(* IEC 61131-3 sources: ST2CPP/examples/projects/robot_arm, 8 files *)

(* ---- math_utils.st ---- *)
(* math_utils.st — 数学工具函数 *)

FUNCTION DEG_TO_RAD : REAL
    VAR_INPUT DEG : REAL; END_VAR
    DEG_TO_RAD := DEG * 3.14159265 / 180.0;
END_FUNCTION

FUNCTION RAD_TO_DEG : REAL
    VAR_INPUT RAD : REAL; END_VAR
    RAD_TO_DEG := RAD * 180.0 / 3.14159265;
END_FUNCTION

FUNCTION CLAMP_REAL : REAL
    VAR_INPUT VAL : REAL; MN : REAL; MX : REAL; END_VAR
    IF VAL > MX THEN
        CLAMP_REAL := MX;
    ELSIF VAL < MN THEN
        CLAMP_REAL := MN;
    ELSE
        CLAMP_REAL := VAL;
    END_IF;
END_FUNCTION

FUNCTION CLAMP_DINT : DINT
    VAR_INPUT VAL : DINT; MN : DINT; MX : DINT; END_VAR
    IF VAL > MX THEN
        CLAMP_DINT := MX;
    ELSIF VAL < MN THEN
        CLAMP_DINT := MN;
    ELSE
        CLAMP_DINT := VAL;
    END_IF;
END_FUNCTION

FUNCTION ABS_REAL : REAL
    VAR_INPUT X : REAL; END_VAR
    IF X < 0.0 THEN
        ABS_REAL := 0.0 - X;
    ELSE
        ABS_REAL := X;
    END_IF;
END_FUNCTION

FUNCTION ABS_DINT : DINT
    VAR_INPUT X : DINT; END_VAR
    IF X < 0 THEN
        ABS_DINT := 0 - X;
    ELSE
        ABS_DINT := X;
    END_IF;
END_FUNCTION

FUNCTION SIGN_REAL : REAL
    VAR_INPUT X : REAL; END_VAR
    IF X > 0.0 THEN
        SIGN_REAL := 1.0;
    ELSIF X < 0.0 THEN
        SIGN_REAL := -1.0;
    ELSE
        SIGN_REAL := 0.0;
    END_IF;
END_FUNCTION

(* 简单梯形速度规划：返回当前周期的目标位置 *)
FUNCTION TRAPZ_POSITION : DINT
    VAR_INPUT
        POS_START   : DINT;     (* 起始位置 *)
        POS_END     : DINT;     (* 目标位置 *)
        VEL_MAX     : DINT;     (* 最大速度 *)
        ACC_MAX     : DINT;     (* 最大加速度 *)
        TIME_MS     : DINT;     (* 已用时间 ms *)
        TOTAL_MS    : DINT;     (* 总时间 ms *)
    END_VAR
    VAR
        DIST        : DINT;
        SIGN_DIR    : DINT;
        ACCEL_TIME  : DINT;
        cruise_time : DINT;
        pos         : DINT;
    END_VAR

    DIST := ABS_DINT(POS_END - POS_START);
    IF POS_END >= POS_START THEN
        SIGN_DIR := 1;
    ELSE
        SIGN_DIR := -1;
    END_IF;

    IF VEL_MAX <= 0 OR ACC_MAX <= 0 OR TOTAL_MS <= 0 THEN
        TRAPZ_POSITION := POS_START;
        RETURN;
    END_IF;

    ACCEL_TIME := VEL_MAX * 1000 / ACC_MAX;
    IF ACCEL_TIME > TOTAL_MS / 2 THEN
        ACCEL_TIME := TOTAL_MS / 2;
    END_IF;

    cruise_time := TOTAL_MS - 2 * ACCEL_TIME;

    IF TIME_MS < ACCEL_TIME THEN
        (* 加速段 *)
        pos := POS_START + SIGN_DIR * ACC_MAX * TIME_MS * TIME_MS / 2000000;
    ELSIF TIME_MS < ACCEL_TIME + cruise_time THEN
        (* 匀速段 *)
        pos := POS_START + SIGN_DIR * (VEL_MAX * ACCEL_TIME / 1000 + VEL_MAX * (TIME_MS - ACCEL_TIME) / 1000);
    ELSIF TIME_MS < TOTAL_MS THEN
        (* 减速段 *)
        pos := POS_END - SIGN_DIR * ACC_MAX * (TOTAL_MS - TIME_MS) * (TOTAL_MS - TIME_MS) / 2000000;
    ELSE
        pos := POS_END;
    END_IF;

    TRAPZ_POSITION := pos;
END_FUNCTION

(* 两点间距离 *)
FUNCTION DISTANCE_3D : REAL
    VAR_INPUT A : POSE_3D; B : POSE_3D; END_VAR
    VAR DX : REAL; DY : REAL; DZ : REAL; END_VAR
    DX := B.X - A.X;
    DY := B.Y - A.Y;
    DZ := B.Z - A.Z;
    DISTANCE_3D := (DX * DX + DY * DY + DZ * DZ);
END_FUNCTION

(* ---- motion_planner.st ---- *)
(* motion_planner.st — 关节空间运动规划器 *)

FUNCTION_BLOCK JOINT_PLANNER
    VAR_INPUT
        TARGET_J    : JOINT_WAYPOINT;   (* 目标关节角度 *)
        SPEED_PCT   : REAL;             (* 速度百分比 0-100 *)
        START       : BOOL;             (* 启动运动 *)
        STOP        : BOOL;             (* 停止运动 *)
        ABORT       : BOOL;             (* 紧急终止 *)
    END_VAR
    VAR_OUTPUT
        CMD_J       : JOINT_WAYPOINT;   (* 当前周期命令 *)
        DONE        : BOOL;             (* 运动完成 *)
        MOVING      : BOOL;             (* 运动中 *)
        PROGRESS    : REAL;             (* 进度 0-100 *)
        ERROR       : BOOL;
        ERROR_CODE  : INT;
    END_VAR
    VAR
        STATE       : INT := 0;         (* 0=Idle, 1=Planning, 2=Moving, 3=Done *)
        START_J     : JOINT_WAYPOINT;   (* 起始关节角度 *)
        TIME_MS     : DINT := 0;
        TOTAL_MS    : DINT := 0;
        SPEED_SCALE : REAL;
        I           : INT;
        DUR         : DINT;
        MAX_DUR     : DINT;
    END_VAR

    IF ABORT THEN
        STATE := 0;
        MOVING := FALSE;
        DONE := FALSE;
        ERROR := TRUE;
        ERROR_CODE := 99;
        RETURN;
    END_IF;

    IF STOP AND STATE = 2 THEN
        STATE := 0;
        MOVING := FALSE;
        DONE := FALSE;
        RETURN;
    END_IF;

    CASE STATE OF
        0:
            (* Idle *)
            DONE := FALSE;
            MOVING := FALSE;
            PROGRESS := 0.0;
            ERROR := FALSE;
            ERROR_CODE := 0;
            IF START THEN
                STATE := 1;
                TIME_MS := 0;
                MAX_DUR := 0;
                SPEED_SCALE := SPEED_PCT / 100.0;
                IF SPEED_SCALE < 0.1 THEN
                    SPEED_SCALE := 0.1;
                END_IF;
                IF SPEED_SCALE > 1.0 THEN
                    SPEED_SCALE := 1.0;
                END_IF;
            END_IF;

        1:
            (* Planning — 计算运动时间 *)
            (* J1 *)
            DUR := ABS_DINT(TARGET_J.J1 * 100);
            IF DUR > MAX_DUR THEN MAX_DUR := DUR; END_IF;
            (* J2 *)
            DUR := ABS_DINT(TARGET_J.J2 * 100);
            IF DUR > MAX_DUR THEN MAX_DUR := DUR; END_IF;
            (* J3 *)
            DUR := ABS_DINT(TARGET_J.J3 * 100);
            IF DUR > MAX_DUR THEN MAX_DUR := DUR; END_IF;
            (* J4 *)
            DUR := ABS_DINT(TARGET_J.J4 * 100);
            IF DUR > MAX_DUR THEN MAX_DUR := DUR; END_IF;
            (* J5 *)
            DUR := ABS_DINT(TARGET_J.J5 * 100);
            IF DUR > MAX_DUR THEN MAX_DUR := DUR; END_IF;
            (* J6 *)
            DUR := ABS_DINT(TARGET_J.J6 * 100);
            IF DUR > MAX_DUR THEN MAX_DUR := DUR; END_IF;

            TOTAL_MS := MAX_DUR * 10 / SPEED_SCALE + 500;
            IF TOTAL_MS < 100 THEN TOTAL_MS := 100; END_IF;
            IF TOTAL_MS > 5000 THEN TOTAL_MS := 5000; END_IF;

            START_J.J1 := CMD_J.J1;
            START_J.J2 := CMD_J.J2;
            START_J.J3 := CMD_J.J3;
            START_J.J4 := CMD_J.J4;
            START_J.J5 := CMD_J.J5;
            START_J.J6 := CMD_J.J6;

            STATE := 2;
            MOVING := TRUE;

        2:
            (* Moving — 每个周期更新 *)
            TIME_MS := TIME_MS + 10;

            CMD_J.J1 := TRAPZ_POSITION(START_J.J1, TARGET_J.J1, 1000, 200, TIME_MS, TOTAL_MS);
            CMD_J.J2 := TRAPZ_POSITION(START_J.J2, TARGET_J.J2, 800, 150, TIME_MS, TOTAL_MS);
            CMD_J.J3 := TRAPZ_POSITION(START_J.J3, TARGET_J.J3, 800, 150, TIME_MS, TOTAL_MS);
            CMD_J.J4 := TRAPZ_POSITION(START_J.J4, TARGET_J.J4, 1200, 300, TIME_MS, TOTAL_MS);
            CMD_J.J5 := TRAPZ_POSITION(START_J.J5, TARGET_J.J5, 1200, 300, TIME_MS, TOTAL_MS);
            CMD_J.J6 := TRAPZ_POSITION(START_J.J6, TARGET_J.J6, 1500, 400, TIME_MS, TOTAL_MS);

            IF TOTAL_MS > 0 THEN
                PROGRESS := TIME_MS * 100.0 / TOTAL_MS;
            END_IF;
            IF PROGRESS > 100.0 THEN PROGRESS := 100.0; END_IF;

            IF TIME_MS >= TOTAL_MS THEN
                CMD_J.J1 := TARGET_J.J1;
                CMD_J.J2 := TARGET_J.J2;
                CMD_J.J3 := TARGET_J.J3;
                CMD_J.J4 := TARGET_J.J4;
                CMD_J.J5 := TARGET_J.J5;
                CMD_J.J6 := TARGET_J.J6;
                STATE := 3;
                MOVING := FALSE;
                DONE := TRUE;
                PROGRESS := 100.0;
            END_IF;

        3:
            (* Done *)
            MOVING := FALSE;
            IF NOT START THEN
                STATE := 0;
                DONE := FALSE;
            END_IF;
    END_CASE;
END_FUNCTION_BLOCK

(* ---- robot_ctrl.st ---- *)
(* robot_ctrl.st — 6轴机械臂主控制器 *)

FUNCTION_BLOCK ROBOT_CTRL
    VAR_INPUT
        START           : BOOL;
        STOP            : BOOL;
        HOME_CMD        : BOOL;
        AUTO_MODE       : BOOL;
        TEACH_MODE      : BOOL;
        SPEED_OVERRIDE  : REAL;          (* 速度倍率 0-100% *)
    END_VAR
    VAR_OUTPUT
        STATE_OUT       : INT;           (* 0=Disabled, 1=Idle, 2=Running, 3=Homing, 4=Error *)
        FAULT           : BOOL;
        FAULT_CODE      : INT;
        HOME_DONE       : BOOL;
        STEP_NUM        : INT;
        CYCLE_COUNT     : DINT;
    END_VAR
    VAR
        (* 6轴伺服 *)
        Srv             : ARRAY[0..5] OF SERVO_CTRL;

        (* 运动规划器 *)
        Planner         : JOINT_PLANNER;

        (* 安全监控 *)
        SafetyMon       : SAFETY_MONITOR;

        (* 关节限位 [轴号][0=下限,1=上限] *)
        JOINT_LIM       : ARRAY[0..5, 0..1] OF DINT;

        (* 伺服状态 *)
        SrvReady        : ARRAY[0..5] OF BOOL;
        SrvFaultArr     : ARRAY[0..5] OF BOOL;
        ActPosArr       : ARRAY[0..5] OF DINT;

        (* 工序步 *)
        PROG_STEP       : INT := 0;
        STEP_ACTIVE     : BOOL := FALSE;
        ALL_DONE        : BOOL := FALSE;

        (* 工序定义：抓取-放置 *)
        GRAB_POS        : JOINT_WAYPOINT := (J1 := 0.0, J2 := -45.0, J3 := 90.0, J4 := 0.0, J5 := 45.0, J6 := 0.0, SPEED := 50.0, DWELL_MS := 500);
        PRE_GRAB_POS    : JOINT_WAYPOINT := (J1 := 0.0, J2 := -20.0, J3 := 45.0, J4 := 0.0, J5 := 20.0, J6 := 0.0, SPEED := 30.0, DWELL_MS := 200);
        HOME_POS        : JOINT_WAYPOINT := (J1 := 0.0, J2 := 0.0, J3 := 0.0, J4 := 0.0, J5 := 0.0, J6 := 0.0, SPEED := 20.0, DWELL_MS := 0);
        PLACE_POS       : JOINT_WAYPOINT := (J1 := 90.0, J2 := -30.0, J3 := 60.0, J4 := 0.0, J5 := 30.0, J6 := 90.0, SPEED := 40.0, DWELL_MS := 300);
        RETRACT_POS     : JOINT_WAYPOINT := (J1 := 90.0, J2 := 0.0, J3 := 0.0, J4 := 0.0, J5 := 0.0, J6 := 0.0, SPEED := 50.0, DWELL_MS := 200);

        (* 辅助 *)
        I               : INT;
        SRV_EN          : ARRAY[0..5] OF BOOL;
        START_PREV      : BOOL := FALSE;
        TRIG_START      : BOOL;
        HOME_PREV       : BOOL := FALSE;
        TRIG_HOME       : BOOL;
        DWELL_TIMER     : INT := 0;
        DWELL_TARGET    : INT := 0;
    END_VAR

    TRIG_START := START AND NOT START_PREV;
    START_PREV := START;
    TRIG_HOME := HOME_CMD AND NOT HOME_PREV;
    HOME_PREV := HOME_CMD;

    (* ─── 关节限位初始化 ─── *)
    JOINT_LIM[0, 0] := -170000;
    JOINT_LIM[0, 1] := 170000;
    JOINT_LIM[1, 0] := -120000;
    JOINT_LIM[1, 1] := 120000;
    JOINT_LIM[2, 0] := -150000;
    JOINT_LIM[2, 1] := 150000;
    JOINT_LIM[3, 0] := -180000;
    JOINT_LIM[3, 1] := 180000;
    JOINT_LIM[4, 0] := -120000;
    JOINT_LIM[4, 1] := 120000;
    JOINT_LIM[5, 0] := -360000;
    JOINT_LIM[5, 1] := 360000;

    (* ─── 速度倍率钳位 ─── *)
    SPEED_OVERRIDE := CLAMP_REAL(SPEED_OVERRIDE, 5.0, 100.0);

    (* ─── 使能所有伺服 ─── *)
    FOR I := 0 TO 5 DO
        SRV_EN[I] := START AND NOT FAULT;
    END_FOR;

    (* ─── 执行伺服控制 ─── *)
    FOR I := 0 TO 5 DO
        Srv[I](
            AXIS_ID := I,
            CMD_POSITION := Planner.CMD_J.J1,
            CMD_MODE := 0,
            ENABLE := SRV_EN[I],
            HOME_CMD := TRIG_HOME,
            RESET_CMD := FALSE,
            VEL_LIMIT := 2000,
            TORQ_LIMIT := 80
        );
        SrvReady[I] := Srv[I].READY;
        SrvFaultArr[I] := Srv[I].FAULT;
        ActPosArr[I] := Srv[I].ACT_POSITION;
    END_FOR;

    (* ─── 安全监控 ─── *)
    SafetyMon(
        E_STOP_IN := EStop,
        SERVO_READY := SrvReady,
        SERVO_FAULT := SrvFaultArr,
        ACT_POSITIONS := ActPosArr,
        JOINT_LIMITS := JOINT_LIM,
        CFG := Safety
    );

    FAULT := NOT SafetyMon.SAFE_OK;
    FAULT_CODE := SafetyMon.ALARM_OUT.ALARM_CODE;

    (* ─── 运动规划器 ─── *)
    Planner(
        SPEED_PCT := SPEED_OVERRIDE,
        STOP := STOP,
        ABORT := FAULT
    );

    (* ─── 主状态机 ─── *)
    CASE STATE_OUT OF
        0:
            (* Disabled *)
            HOME_DONE := FALSE;
            PROG_STEP := 0;
            STEP_ACTIVE := FALSE;
            ALL_DONE := FALSE;
            IF START AND SafetyMon.SAFE_OK THEN
                STATE_OUT := 1;
            END_IF;

        1:
            (* Idle — 等待启动 *)
            IF NOT START THEN
                STATE_OUT := 0;
            END_IF;

            IF TRIG_HOME AND NOT HOME_DONE THEN
                STATE_OUT := 3;
            END_IF;

            IF AUTO_MODE AND HOME_DONE AND TRIG_START THEN
                STATE_OUT := 2;
                PROG_STEP := 0;
                STEP_ACTIVE := FALSE;
                ALL_DONE := FALSE;
                CYCLE_COUNT := 0;
            END_IF;

        2:
            (* Running — 执行工序 *)
            IF STOP OR FAULT THEN
                STATE_OUT := 1;
                Planner.STOP := TRUE;
            END_IF;

            IF NOT STEP_ACTIVE THEN
                CASE PROG_STEP OF
                    0:
                        (* 安全位 *)
                        Planner.TARGET_J := PRE_GRAB_POS;
                        Planner.START := TRUE;
                        STEP_ACTIVE := TRUE;
                        DWELL_TIMER := 0;
                        DWELL_TARGET := PRE_GRAB_POS.DWELL_MS;

                    1:
                        (* 抓取位 *)
                        Planner.TARGET_J := GRAB_POS;
                        Planner.START := TRUE;
                        STEP_ACTIVE := TRUE;
                        DWELL_TIMER := 0;
                        DWELL_TARGET := GRAB_POS.DWELL_MS;

                    2:
                        (* 抓取后抬升 *)
                        Planner.TARGET_J := PRE_GRAB_POS;
                        Planner.START := TRUE;
                        STEP_ACTIVE := TRUE;
                        DWELL_TIMER := 0;
                        DWELL_TARGET := 200;

                    3:
                        (* 放置位 *)
                        Planner.TARGET_J := PLACE_POS;
                        Planner.START := TRUE;
                        STEP_ACTIVE := TRUE;
                        DWELL_TIMER := 0;
                        DWELL_TARGET := PLACE_POS.DWELL_MS;

                    4:
                        (* 回缩 *)
                        Planner.TARGET_J := RETRACT_POS;
                        Planner.START := TRUE;
                        STEP_ACTIVE := TRUE;
                        DWELL_TIMER := 0;
                        DWELL_TARGET := RETRACT_POS.DWELL_MS;

                    5:
                        (* 回零 *)
                        Planner.TARGET_J := HOME_POS;
                        Planner.START := TRUE;
                        STEP_ACTIVE := TRUE;
                        DWELL_TIMER := 0;
                        DWELL_TARGET := HOME_POS.DWELL_MS;

                    ELSE
                        ALL_DONE := TRUE;
                        CYCLE_COUNT := CYCLE_COUNT + 1;
                        PROG_STEP := 0;
                        STEP_ACTIVE := FALSE;
                END_CASE;
            ELSE
                Planner.START := FALSE;
                IF Planner.DONE THEN
                    DWELL_TIMER := DWELL_TIMER + 10;
                    IF DWELL_TIMER >= DWELL_TARGET THEN
                        PROG_STEP := PROG_STEP + 1;
                        STEP_ACTIVE := FALSE;
                    END_IF;
                END_IF;
            END_IF;

            STEP_NUM := PROG_STEP;

        3:
            (* Homing *)
            Planner.TARGET_J := HOME_POS;
            Planner.SPEED_PCT := 20.0;
            Planner.START := TRUE;

            IF Planner.DONE THEN
                HOME_DONE := TRUE;
                STATE_OUT := 1;
                Planner.START := FALSE;
            END_IF;

        4:
            (* Error *)
            IF NOT FAULT AND START THEN
                STATE_OUT := 0;
            END_IF;
    END_CASE;

    (* ─── 故障跳转 ─── *)
    IF FAULT AND STATE_OUT <> 4 THEN
        STATE_OUT := 4;
        Planner.ABORT := TRUE;
    END_IF;
END_FUNCTION_BLOCK

(* ---- safety.st ---- *)
(* safety.st — 安全监控功能块 *)

FUNCTION_BLOCK SAFETY_MONITOR
    VAR_INPUT
        E_STOP_IN       : BOOL;         (* 急停输入 *)
        SERVO_READY     : ARRAY[0..5] OF BOOL;
        SERVO_FAULT     : ARRAY[0..5] OF BOOL;
        ACT_POSITIONS   : ARRAY[0..5] OF DINT;
        JOINT_LIMITS    : ARRAY[0..5, 0..1] OF DINT;  (* [轴号][0=下限,1=上限] *)
        CFG             : SAFETY_CFG;
    END_VAR
    VAR_OUTPUT
        SAFE_OK         : BOOL;         (* 安全状态正常 *)
        ALARM_OUT       : SAFETY_ALARM;
        ALL_SERVO_OK    : BOOL;
        SPEED_OK        : BOOL;
        LIMITS_OK       : BOOL;
    END_VAR
    VAR
        I               : INT;
        J               : INT;
        OVERTRAVEL      : BOOL;
        SRV_FAULT_ANY   : BOOL;
        SRV_NOT_READY   : BOOL;
    END_VAR

    (* ─── 急停检测 ─── *)
    ALARM_OUT.E_STOP := NOT E_STOP_IN;
    IF CFG.E_STOP_ACTIVE AND ALARM_OUT.E_STOP THEN
        ALARM_OUT.ALARM_CODE := 1;
    END_IF;

    (* ─── 伺服故障/就绪检测 ─── *)
    SRV_FAULT_ANY := FALSE;
    SRV_NOT_READY := FALSE;
    FOR I := 0 TO 5 DO
        IF SERVO_FAULT[I] THEN
            SRV_FAULT_ANY := TRUE;
        END_IF;
        IF NOT SERVO_READY[I] THEN
            SRV_NOT_READY := TRUE;
        END_IF;
    END_FOR;

    ALARM_OUT.SERVO_FAULT := SRV_FAULT_ANY;
    ALARM_OUT.COMM_LOST := SRV_NOT_READY;
    ALL_SERVO_OK := NOT SRV_FAULT_ANY AND NOT SRV_NOT_READY;

    (* ─── 关节软限位检测 ─── *)
    OVERTRAVEL := FALSE;
    IF CFG.JOINT_LIMITS_EN THEN
        FOR I := 0 TO 5 DO
            IF ACT_POSITIONS[I] < JOINT_LIMITS[I, 0] THEN
                OVERTRAVEL := TRUE;
            END_IF;
            IF ACT_POSITIONS[I] > JOINT_LIMITS[I, 1] THEN
                OVERTRAVEL := TRUE;
            END_IF;
        END_FOR;
    END_IF;
    ALARM_OUT.JOINT_OVERTRAVEL := OVERTRAVEL;
    LIMITS_OK := NOT OVERTRAVEL;

    (* ─── 速度/扭矩限制（通过全局速度百分比） ─── *)
    SPEED_OK := TRUE;

    (* ─── 碰撞检测（简化：任意轴扭矩超限） ─── *)
    ALARM_OUT.COLLISION := FALSE;
    ALARM_OUT.OVERSPEED := FALSE;
    ALARM_OUT.WORKSPACE_VIOL := FALSE;

    (* ─── 综合安全状态 ─── *)
    SAFE_OK := NOT ALARM_OUT.E_STOP
               AND NOT ALARM_OUT.SERVO_FAULT
               AND NOT ALARM_OUT.JOINT_OVERTRAVEL
               AND NOT ALARM_OUT.COMM_LOST
               AND NOT ALARM_OUT.COLLISION;

    ALARM_OUT.ALARM_CODE := 0;
    IF ALARM_OUT.E_STOP THEN ALARM_OUT.ALARM_CODE := 1; END_IF;
    IF ALARM_OUT.SERVO_FAULT THEN ALARM_OUT.ALARM_CODE := 2; END_IF;
    IF ALARM_OUT.JOINT_OVERTRAVEL THEN ALARM_OUT.ALARM_CODE := 3; END_IF;
    IF ALARM_OUT.COMM_LOST THEN ALARM_OUT.ALARM_CODE := 4; END_IF;
    IF ALARM_OUT.COLLISION THEN ALARM_OUT.ALARM_CODE := 5; END_IF;
    IF ALARM_OUT.OVERSPEED THEN ALARM_OUT.ALARM_CODE := 6; END_IF;
    IF ALARM_OUT.WORKSPACE_VIOL THEN ALARM_OUT.ALARM_CODE := 7; END_IF;
END_FUNCTION_BLOCK

(* ---- servo_drive.st ---- *)
(* servo_drive.st — 单轴伺服驱动器控制功能块 *)

FUNCTION_BLOCK SERVO_CTRL
    VAR_INPUT
        AXIS_ID         : INT;          (* 轴号 0-5 *)
        CMD_POSITION    : DINT;         (* 命令位置 *)
        CMD_MODE        : INT;          (* 0=位置, 1=速度, 2=扭矩 *)
        ENABLE          : BOOL;         (* 使能 *)
        HOME_CMD        : BOOL;         (* 回原点命令 *)
        RESET_CMD       : BOOL;         (* 故障复位 *)
        VEL_LIMIT      : DINT;         (* 速度限制 *)
        TORQ_LIMIT     : INT;          (* 扭矩限制 *)
    END_VAR
    VAR_OUTPUT
        ACT_POSITION    : DINT;         (* 实际位置 *)
        ACT_VELOCITY    : DINT;         (* 实际速度 *)
        ACT_TORQUE      : INT;          (* 实际扭矩 *)
        IN_POSITION     : BOOL;         (* 到位 *)
        READY           : BOOL;         (* 准备就绪 *)
        FAULT           : BOOL;         (* 故障 *)
        HOMED           : BOOL;         (* 已回原点 *)
        ERROR_CODE      : WORD;         (* 故障码 *)
    END_VAR
    VAR
        STATE           : INT := 0;     (* 0=Disabled, 1=Enabling, 2=Enabled, 3=Fault *)
        CMD_CTRL        : WORD;
        IN_POS_COUNT    : INT := 0;
        HOME_STATE      : INT := 0;
        PREV_RESET      : BOOL := FALSE;
        TRIG_RESET      : BOOL;
        FAULT_LATCH     : BOOL := FALSE;
        READY_DELAY     : INT := 0;
    END_VAR

    (* ─── 读取硬件状态 ─── *)
    IF AXIS_ID = 0 THEN
        ACT_POSITION := Srv1ActPos;
        ACT_VELOCITY := Srv1ActVel;
        ACT_TORQUE := Srv1ActTorq;
        ERROR_CODE := Srv1Status;
    ELSIF AXIS_ID = 1 THEN
        ACT_POSITION := Srv2ActPos;
        ACT_VELOCITY := Srv2ActVel;
        ACT_TORQUE := Srv2ActTorq;
        ERROR_CODE := Srv2Status;
    ELSIF AXIS_ID = 2 THEN
        ACT_POSITION := Srv3ActPos;
        ACT_VELOCITY := Srv3ActVel;
        ACT_TORQUE := Srv3ActTorq;
        ERROR_CODE := Srv3Status;
    ELSIF AXIS_ID = 3 THEN
        ACT_POSITION := Srv4ActPos;
        ACT_VELOCITY := Srv4ActVel;
        ACT_TORQUE := Srv4ActTorq;
        ERROR_CODE := Srv4Status;
    ELSIF AXIS_ID = 4 THEN
        ACT_POSITION := Srv5ActPos;
        ACT_VELOCITY := Srv5ActVel;
        ACT_TORQUE := Srv5ActTorq;
        ERROR_CODE := Srv5Status;
    ELSE
        ACT_POSITION := Srv6ActPos;
        ACT_VELOCITY := Srv6ActVel;
        ACT_TORQUE := Srv6ActTorq;
        ERROR_CODE := Srv6Status;
    END_IF;

    (* ─── 故障检测 ─── *)
    IF ERROR_CODE <> 0 THEN
        FAULT := TRUE;
        FAULT_LATCH := TRUE;
        STATE := 3;
    END_IF;

    (* ─── 故障复位 ─── *)
    TRIG_RESET := RESET_CMD AND NOT PREV_RESET;
    PREV_RESET := RESET_CMD;
    IF TRIG_RESET AND FAULT_LATCH THEN
        FAULT_LATCH := FALSE;
        FAULT := FALSE;
        ERROR_CODE := 0;
        STATE := 0;
    END_IF;

    (* ─── 状态机 ─── *)
    CASE STATE OF
        0:
            (* Disabled *)
            READY := FALSE;
            HOMED := FALSE;
            CMD_CTRL := 0;
            IF ENABLE AND NOT FAULT_LATCH THEN
                STATE := 1;
                READY_DELAY := 0;
            END_IF;

        1:
            (* Enabling — 等待驱动器就绪 *)
            READY_DELAY := READY_DELAY + 1;
            CMD_CTRL := 16#0007;       (* 使能 + 位置模式 *)
            IF READY_DELAY >= 10 THEN
                STATE := 2;
                READY := TRUE;
            END_IF;

        2:
            (* Enabled *)
            READY := TRUE;
            CMD_CTRL := 16#000F;       (* 使能 + 位置模式 + 运行 *)

            IF NOT ENABLE THEN
                STATE := 0;
                READY := FALSE;
            END_IF;

            (* 回原点 *)
            IF HOME_CMD THEN
                HOME_STATE := 1;
            END_IF;

            IF HOME_STATE = 1 THEN
                CMD_CTRL := 16#001F;   (* 回原点模式 *)
                IF HomeSwitch THEN
                    CMD_CTRL := 16#002F;   (* 原点锁定 *)
                    HOME_STATE := 2;
                END_IF;
            ELSIF HOME_STATE = 2 THEN
                CMD_CTRL := 16#002F;
                HOME_STATE := 3;
            ELSIF HOME_STATE = 3 THEN
                HOMED := TRUE;
                HOME_STATE := 0;
            END_IF;

        3:
            (* Fault *)
            READY := FALSE;
            CMD_CTRL := 0;
            IF NOT FAULT_LATCH THEN
                STATE := 0;
            END_IF;
    END_CASE;

    (* ─── 到位判断 ─── *)
    IF ABS_DINT(ACT_POSITION - CMD_POSITION) < 100 THEN
        IN_POS_COUNT := IN_POS_COUNT + 1;
        IF IN_POS_COUNT >= 5 THEN
            IN_POSITION := TRUE;
        END_IF;
    ELSE
        IN_POS_COUNT := 0;
        IN_POSITION := FALSE;
    END_IF;

    (* ─── 写入控制字和命令 ─── *)
    IF AXIS_ID = 0 THEN
        Srv1Ctrl := CMD_CTRL;
        Srv1CmdPos := CMD_POSITION;
    ELSIF AXIS_ID = 1 THEN
        Srv2Ctrl := CMD_CTRL;
        Srv2CmdPos := CMD_POSITION;
    ELSIF AXIS_ID = 2 THEN
        Srv3Ctrl := CMD_CTRL;
        Srv3CmdPos := CMD_POSITION;
    ELSIF AXIS_ID = 3 THEN
        Srv4Ctrl := CMD_CTRL;
        Srv4CmdPos := CMD_POSITION;
    ELSIF AXIS_ID = 4 THEN
        Srv5Ctrl := CMD_CTRL;
        Srv5CmdPos := CMD_POSITION;
    ELSE
        Srv6Ctrl := CMD_CTRL;
        Srv6CmdPos := CMD_POSITION;
    END_IF;
END_FUNCTION_BLOCK

(* ---- io_config.st ---- *)
(* io_config.st — 6轴机械臂 EtherCAT I/O 映射 *)

VAR_GLOBAL
    (* ─── EtherCAT 伺服驱动器 PDO（6 轴） ─── *)

    (* 轴1-3：基座/大臂/小臂（高扭矩） *)
    Srv1CmdPos     AT %ID0   : DINT;      (* 命令位置 *)
    Srv1Status     AT %IW0   : WORD;      (* 状态字 *)
    Srv1ActPos     AT %ID4   : DINT;      (* 实际位置 *)
    Srv1ActVel     AT %ID8   : DINT;      (* 实际速度 *)
    Srv1ActTorq    AT %IW4   : INT;       (* 实际扭矩 *)
    Srv1Ctrl       AT %QW0   : WORD;      (* 控制字 *)
    Srv1CmdVel     AT %QD0   : DINT;      (* 命令速度 *)
    Srv1CmdTorq    AT %QW2   : INT;       (* 命令扭矩 *)

    Srv2CmdPos     AT %ID12  : DINT;
    Srv2Status     AT %IW8   : WORD;
    Srv2ActPos     AT %ID16  : DINT;
    Srv2ActVel     AT %ID20  : DINT;
    Srv2ActTorq    AT %IW10  : INT;
    Srv2Ctrl       AT %QW4   : WORD;
    Srv2CmdVel     AT %QD4   : DINT;
    Srv2CmdTorq    AT %QW6   : INT;

    Srv3CmdPos     AT %ID24  : DINT;
    Srv3Status     AT %IW12  : WORD;
    Srv3ActPos     AT %ID28  : DINT;
    Srv3ActVel     AT %ID32  : DINT;
    Srv3ActTorq    AT %IW14  : INT;
    Srv3Ctrl       AT %QW8   : WORD;
    Srv3CmdVel     AT %QD8   : DINT;
    Srv3CmdTorq    AT %QW10  : INT;

    (* 轴4-6：腕部（小扭矩/高速） *)
    Srv4CmdPos     AT %ID36  : DINT;
    Srv4Status     AT %IW16  : WORD;
    Srv4ActPos     AT %ID40  : DINT;
    Srv4ActVel     AT %ID44  : DINT;
    Srv4ActTorq    AT %IW18  : INT;
    Srv4Ctrl       AT %QW12  : WORD;
    Srv4CmdVel     AT %QD12  : DINT;
    Srv4CmdTorq    AT %QW14  : INT;

    Srv5CmdPos     AT %ID48  : DINT;
    Srv5Status     AT %IW20  : WORD;
    Srv5ActPos     AT %ID52  : DINT;
    Srv5ActVel     AT %ID56  : DINT;
    Srv5ActTorq    AT %IW22  : INT;
    Srv5Ctrl       AT %QW16  : WORD;
    Srv5CmdVel     AT %QD16  : DINT;
    Srv5CmdTorq    AT %QW18  : INT;

    Srv6CmdPos     AT %ID60  : DINT;
    Srv6Status     AT %IW24  : WORD;
    Srv6ActPos     AT %ID64  : DINT;
    Srv6ActVel     AT %ID68  : DINT;
    Srv6ActTorq    AT %IW26  : INT;
    Srv6Ctrl       AT %QW20  : WORD;
    Srv6CmdVel     AT %QD20  : DINT;
    Srv6CmdTorq    AT %QW22  : INT;

    (* ─── 数字量 I/O ─── *)
    StartBtn       AT %IX0.0 : BOOL;      (* 启动按钮 *)
    StopBtn        AT %IX0.1 : BOOL;      (* 停止按钮 *)
    EStop          AT %IX0.2 : BOOL;      (* 急停按钮（NC） *)
    HomeSwitch     AT %IX0.3 : BOOL;      (* 原点开关 *)
    GripSensor     AT %IX0.4 : BOOL;      (* 夹爪力传感器 *)
    PartDetect     AT %IX0.5 : BOOL;      (* 工件检测 *)
    AutoMode       AT %IX0.6 : BOOL;      (* 自动模式 *)
    TeachMode      AT %IX0.7 : BOOL;      (* 示教模式 *)

    RobotRun       AT %QX0.0 : BOOL;      (* 运行指示灯 *)
    RobotError     AT %QX0.1 : BOOL;      (* 故障灯 *)
    RobotHome      AT %QX0.2 : BOOL;      (* 原点灯 *)
    GripperOpen    AT %QX0.3 : BOOL;      (* 夹爪打开 *)
    GripperClose   AT %QX0.4 : BOOL;      (* 夹爪闭合 *)
    ConveyorRun    AT %QX0.5 : BOOL;      (* 传送带运行 *)
    WeldEnable     AT %QX0.6 : BOOL;      (* 焊接使能 *)
    ToolChange     AT %QX0.7 : BOOL;      (* 换刀信号 *)

    (* ─── 模拟量 I/O ─── *)
    WeldCurrent    AT %QW24 : INT;        (* 焊接电流 *)
    WeldVoltage    AT %QW26 : INT;        (* 焊接电压 *)
    ForceSensor    AT %IW28 : INT;        (* 力传感器 *)
    VisionReady    AT %IW30 : INT;        (* 视觉系统状态 *)

    (* ─── 系统全局变量 ─── *)
    RobotEnabled   : BOOL := FALSE;
    HomeDone       : BOOL := FALSE;
    ProgramRunning : BOOL := FALSE;
    CurrentStep    : INT := 0;
    TotalCycles    : DINT := 0;
    CycleTime      : DINT := 0;
    MaxCycleTime   : DINT := 0;

    (* ─── 伺服状态数组 ─── *)
    SrvState       : ARRAY[0..5] OF SERVO_STATE;

    (* ─── 当前位姿 ─── *)
    CurrentPose    : POSE_3D;
    TargetPose     : POSE_3D;

    (* ─── 运动状态 ─── *)
    Motion         : MOTION_STATE;

    (* ─── 安全系统 ─── *)
    Safety         : SAFETY_CFG;
    Alarm          : SAFETY_ALARM;
END_VAR

(* ---- main.st ---- *)
(* main.st — 6轴机械臂主程序 *)

PROGRAM ROBOT_MAIN
    VAR_INPUT
        StartBtn    AT %IX0.0 : BOOL;
        StopBtn     AT %IX0.1 : BOOL;
        EStop       AT %IX0.2 : BOOL;
        HomeSw      AT %IX0.3 : BOOL;
        GripSensor  AT %IX0.4 : BOOL;
        PartDetect  AT %IX0.5 : BOOL;
        AutoMode    AT %IX0.6 : BOOL;
        TeachMode   AT %IX0.7 : BOOL;
    END_VAR
    VAR_OUTPUT
        RunLamp     AT %QX0.0 : BOOL;
        ErrorLamp   AT %QX0.1 : BOOL;
        HomeLamp    AT %QX0.2 : BOOL;
        GripOpen    AT %QX0.3 : BOOL;
        GripClose   AT %QX0.4 : BOOL;
        ConvRun     AT %QX0.5 : BOOL;
        WeldEn      AT %QX0.6 : BOOL;
        ToolChg     AT %QX0.7 : BOOL;
    END_VAR
    VAR
        Robot       : ROBOT_CTRL;
        SpeedOvr    : REAL := 80.0;
        CycleTimeMs : DINT := 0;
        TotalParts  : DINT := 0;
        PartReady   : BOOL := FALSE;
        GripDone    : BOOL := FALSE;
        I           : INT;
    END_VAR

    (* ─── 安全配置 ─── *)
    Safety.E_STOP_ACTIVE := TRUE;
    Safety.JOINT_LIMITS_EN := TRUE;
    Safety.COLLISION_EN := TRUE;
    Safety.SPEED_LIMIT_EN := TRUE;
    Safety.WORKSPACE_EN := TRUE;
    Safety.MAX_SPEED_PCT := 100.0;
    Safety.MAX_TORQUE_PCT := 80.0;

    (* ─── 速度倍率 ─── *)
    SpeedOvr := CLAMP_REAL(SpeedOvr, 5.0, 100.0);

    (* ─── 主控制器调用 ─── *)
    Robot(
        START := StartBtn,
        STOP := StopBtn,
        HOME_CMD := HomeSw,
        AUTO_MODE := AutoMode,
        TEACH_MODE := TeachMode,
        SPEED_OVERRIDE := SpeedOvr
    );

    (* ─── 指示灯 ─── *)
    RunLamp := Robot.STATE_OUT = 2;
    ErrorLamp := Robot.FAULT;
    HomeLamp := Robot.HOME_DONE;

    (* ─── 传送带控制 ─── *)
    IF AutoMode AND PartDetect AND NOT GripDone THEN
        ConvRun := TRUE;
    ELSIF GripDone THEN
        ConvRun := FALSE;
    END_IF;

    (* ─── 夹爪控制 ─── *)
    IF Robot.STATE_OUT = 2 AND Robot.STEP_NUM = 1 THEN
        GripClose := TRUE;
        GripOpen := FALSE;
    ELSIF Robot.STATE_OUT = 2 AND (Robot.STEP_NUM = 3 OR Robot.STEP_NUM = 4) THEN
        GripOpen := TRUE;
        GripClose := FALSE;
    ELSE
        GripOpen := TRUE;
        GripClose := FALSE;
    END_IF;

    (* ─── 焊接使能 ─── *)
    WeldEn := FALSE;

    (* ─── 换刀信号 ─── *)
    ToolChg := FALSE;

    (* ─── 统计 ─── *)
    TotalParts := Robot.CYCLE_COUNT;

    (* ─── 伺服状态采集 ─── *)
    SrvState[0].ENABLED := Robot.Srv[0].READY;
    SrvState[0].FAULT := Robot.Srv[0].FAULT;
    SrvState[0].IN_POSITION := Robot.Srv[0].IN_POSITION;
    SrvState[0].POSITION := Robot.Srv[0].ACT_POSITION;
    SrvState[0].VELOCITY := Robot.Srv[0].ACT_VELOCITY;
    SrvState[0].TORQUE := Robot.Srv[0].ACT_TORQUE;

    SrvState[1].ENABLED := Robot.Srv[1].READY;
    SrvState[1].FAULT := Robot.Srv[1].FAULT;
    SrvState[1].IN_POSITION := Robot.Srv[1].IN_POSITION;
    SrvState[1].POSITION := Robot.Srv[1].ACT_POSITION;
    SrvState[1].VELOCITY := Robot.Srv[1].ACT_VELOCITY;
    SrvState[1].TORQUE := Robot.Srv[1].ACT_TORQUE;

    SrvState[2].ENABLED := Robot.Srv[2].READY;
    SrvState[2].FAULT := Robot.Srv[2].FAULT;
    SrvState[2].IN_POSITION := Robot.Srv[2].IN_POSITION;
    SrvState[2].POSITION := Robot.Srv[2].ACT_POSITION;
    SrvState[2].VELOCITY := Robot.Srv[2].ACT_VELOCITY;
    SrvState[2].TORQUE := Robot.Srv[2].ACT_TORQUE;

    SrvState[3].ENABLED := Robot.Srv[3].READY;
    SrvState[3].FAULT := Robot.Srv[3].FAULT;
    SrvState[3].IN_POSITION := Robot.Srv[3].IN_POSITION;
    SrvState[3].POSITION := Robot.Srv[3].ACT_POSITION;
    SrvState[3].VELOCITY := Robot.Srv[3].ACT_VELOCITY;
    SrvState[3].TORQUE := Robot.Srv[3].ACT_TORQUE;

    SrvState[4].ENABLED := Robot.Srv[4].READY;
    SrvState[4].FAULT := Robot.Srv[4].FAULT;
    SrvState[4].IN_POSITION := Robot.Srv[4].IN_POSITION;
    SrvState[4].POSITION := Robot.Srv[4].ACT_POSITION;
    SrvState[4].VELOCITY := Robot.Srv[4].ACT_VELOCITY;
    SrvState[4].TORQUE := Robot.Srv[4].ACT_TORQUE;

    SrvState[5].ENABLED := Robot.Srv[5].READY;
    SrvState[5].FAULT := Robot.Srv[5].FAULT;
    SrvState[5].IN_POSITION := Robot.Srv[5].IN_POSITION;
    SrvState[5].POSITION := Robot.Srv[5].ACT_POSITION;
    SrvState[5].VELOCITY := Robot.Srv[5].ACT_VELOCITY;
    SrvState[5].TORQUE := Robot.Srv[5].ACT_TORQUE;

    (* ─── 周期统计 ─── *)
    TotalCycles := TotalCycles + 1;
    CycleTime := CycleTimeMs;
    IF CycleTimeMs > MaxCycleTime THEN
        MaxCycleTime := CycleTimeMs;
    END_IF;

    Motion.STATE := Robot.STATE_OUT;
    Motion.PROGRESS := Robot.Planner.PROGRESS;
    CurrentStep := Robot.STEP_NUM;
    HomeDone := Robot.HOME_DONE;
    ProgramRunning := Robot.STATE_OUT = 2;
    RobotEnabled := Robot.STATE_OUT <> 0;
    RobotRun := ProgramRunning;
    RobotError := Robot.FAULT;
    RobotHome := HomeDone;
END_PROGRAM

(* ---- types.st ---- *)
(* types.st — 6轴机械臂类型定义 *)

TYPE
    (* 伺服驱动器状态 *)
    SERVO_STATE :
    STRUCT
        POSITION    : DINT;      (* 编码器位置，单位: 脉冲 *)
        VELOCITY    : DINT;      (* 当前速度，单位: 脉冲/周期 *)
        TORQUE      : INT;       (* 当前扭矩，单位: 额定扭矩百分比 *)
        STATUS      : WORD;      (* 状态字 *)
        ERROR_CODE  : WORD;      (* 故障码 *)
        ENABLED     : BOOL;      (* 使能状态 *)
        IN_POSITION : BOOL;      (* 到位信号 *)
        FAULT       : BOOL;      (* 故障标志 *)
    END_STRUCT;

    (* 关节配置 *)
    JOINT_CFG :
    STRUCT
        JOINT_NAME      : INT;         (* 关节名称编号 *)
        JOINT_TYPE      : INT;         (* 0=旋转, 1=移动 *)
        GEAR_RATIO      : REAL;        (* 减速比 *)
        PULSES_PER_REV  : DINT;        (* 编码器每转脉冲数 *)
        POS_MIN         : DINT;        (* 正向软限位 *)
        POS_MAX         : DINT;        (* 反向软限位 *)
        VEL_MAX         : DINT;        (* 最大速度 *)
        ACC_MAX         : DINT;        (* 最大加速度 *)
        HOME_OFFSET     : DINT;        (* 零点偏移 *)
        DIRECTION       : INT;         (* 1=正向, -1=反向 *)
    END_STRUCT;

    (* DH 参数（Denavit-Hartenberg） *)
    DH_PARAM :
    STRUCT
        A       : REAL;        (* 连杆长度 mm *)
        ALPHA   : REAL;        (* 连杆扭角 rad *)
        D       : REAL;        (* 连杆偏距 mm *)
        THETA   : REAL;        (* 关节角度 rad *)
    END_STRUCT;

    (* 3D 位姿 *)
    POSE_3D :
    STRUCT
        X   : REAL;            (* X 坐标 mm *)
        Y   : REAL;            (* Y 坐标 mm *)
        Z   : REAL;            (* Z 坐标 mm *)
        RX  : REAL;            (* 旋转 X rad *)
        RY  : REAL;            (* 旋转 Y rad *)
        RZ  : REAL;            (* 旋转 Z rad *)
    END_STRUCT;

    (* 轨迹点 *)
    WAYPOINT :
    STRUCT
        POSE        : POSE_3D;
        SPEED       : REAL;        (* 速度百分比 0-100 *)
        BLEND_R     : REAL;        (* 轨迹过渡半径 mm *)
        DWELL_MS    : INT;         (* 停留时间 ms *)
    END_STRUCT;

    (* 关节空间轨迹点 *)
    JOINT_WAYPOINT :
    STRUCT
        J1      : REAL;            (* 关节1角度 deg *)
        J2      : REAL;
        J3      : REAL;
        J4      : REAL;
        J5      : REAL;
        J6      : REAL;
        SPEED   : REAL;
        DWELL_MS : INT;
    END_STRUCT;

    (* 运动状态 *)
    MOTION_STATE :
    STRUCT
        TARGET      : POSE_3D;
        CURRENT     : POSE_3D;
        ERROR       : POSE_3D;
        JOINT_TARGET : JOINT_WAYPOINT;
        JOINT_CURRENT : JOINT_WAYPOINT;
        STATE       : INT;         (* 0=空闲, 1=运动中, 2=到位, 3=暂停, 4=错误 *)
        PROGRESS    : REAL;        (* 运动进度 0-100% *)
        TOTAL_TIME  : DINT;        (* 总运行时间 ms *)
        ERR_MSG     : INT;         (* 错误码 *)
    END_STRUCT;

    (* 安全参数 *)
    SAFETY_CFG :
    STRUCT
        E_STOP_ACTIVE     : BOOL;
        JOINT_LIMITS_EN   : BOOL;
        COLLISION_EN      : BOOL;
        SPEED_LIMIT_EN    : BOOL;
        WORKSPACE_EN      : BOOL;
        MAX_SPEED_PCT     : REAL;        (* 全局速度限制 % *)
        MAX_TORQUE_PCT    : REAL;        (* 全局扭矩限制 % *)
    END_STRUCT;

    (* 安全告警 *)
    SAFETY_ALARM :
    STRUCT
        E_STOP          : BOOL;
        JOINT_OVERTRAVEL : BOOL;
        COLLISION       : BOOL;
        OVERSPEED       : BOOL;
        WORKSPACE_VIOL  : BOOL;
        SERVO_FAULT     : BOOL;
        COMM_LOST       : BOOL;
        ALARM_CODE      : INT;
    END_STRUCT;

    (* 程序段 *)
    PROGRAM_SEGMENT :
    STRUCT
        SEG_TYPE    : INT;         (* 0=关节运动, 1=直线运动, 2=圆弧, 3=IO操作, 4=延时 *)
        TARGET      : JOINT_WAYPOINT;
        LINEAR_TARGET : POSE_3D;
        SPEED_PCT   : REAL;
        IO_CMD      : INT;         (* IO 操作编号 *)
        IO_VALUE    : BOOL;        (* IO 值 *)
        DELAY_MS    : INT;
        ENABLED     : BOOL;
    END_STRUCT;
END_TYPE
